// TIA Portal V20 export
VAR_GLOBAL   // PLC tag table "ENTRANCE"
   btnEmStopCraneEntCUCh1 AT %I500.0 : Bool;   // Emergency stop Crane entrance control panel Channel 1
   craneEntCUCraneOnKeyCh1 AT %I500.1 : Bool;   // Crane ON key switch Crane entrance control panel Channel 1
   mhOverloadBypassKeyCh1 AT %I500.2 : Bool;   // MH overload bypass key switch Channel 1
   craneMovementsProhibitionCh1 AT %I500.3 : Bool;   // Crane movements prohibition switch Channel 1
   btnEmStopCraneEntCUCh2 AT %I500.4 : Bool;   // Emergency stop Crane entrance control panel Channel 2
   craneEntCUCraneOnKeyCh2 AT %I500.5 : Bool;   // Crane ON key switch Crane entrance control panel Channel 2
   mhOverloadBypassKeyCh2 AT %I500.6 : Bool;   // MH overload bypass key switch Channel 2
   craneMovementsProhibitionCh2 AT %I500.7 : Bool;   // Crane movements prohibition switch Channel 2
   btnEmStopCraneEntCUCh1VS AT %I501.0 : Bool;   // Emergency stop Crane entrance control panel Channel 1 Supply
   craneEntCUCraneOnKeyCh1VS AT %I501.1 : Bool;   // Crane ON key switch Crane entrance control panel Channel 1 Supply
   mhOverloadBypassKeyCh1VS AT %I501.2 : Bool;   // MH overload bypass key switch Channel 1 Supply
   craneMovementsProhibitionCh1VS AT %I501.3 : Bool;   // Crane movements prohibition switch Channel 1 Supply
   btnEmStopCraneEntCUCh2VS AT %I501.4 : Bool;   // Emergency stop Crane entrance control panel Channel 2 Supply
   craneEntCUCraneOnKeyCh2VS AT %I501.5 : Bool;   // Crane ON key switch Crane entrance control panel Channel 2 Supply
   mhOverloadBypassKeyCh2VS AT %I501.6 : Bool;   // MH overload bypass key switch Channel 2 Supply
   craneMovementsProhibitionCh2VS AT %I501.7 : Bool;   // Crane movements prohibition switch Channel 2 Supply
   craneEntCUOpModeRCOS AT %I550.0 : Bool;   // Crane entrance control panel Operation mode RCOS
   craneEntCUOpModeCabin AT %I550.1 : Bool;   // Crane entrance control panel Operation mode Cabin
   craneEntCUOpModeRadio AT %I550.2 : Bool;   // Crane entrance control panel Operation mode Radio station
   craneEntCUOpModeGround AT %I550.3 : Bool;   // Crane entrance control panel Operation mode Ground level control
   craneEntCUOpModeSpare AT %I550.4 : Bool;   // Crane entrance control panel Operation mode Spare
   craneEntCUCraneOn AT %I550.5 : Bool;   // Crane entrance control panel Crane ON
   craneEntCUCraneOff AT %I550.6 : Bool;   // Crane entrance control panel Crane OFF
   craneEntCUFaultReset AT %I550.7 : Bool;   // Crane entrance control panel Fault reset
   craneEntCULampTest AT %I551.0 : Bool;   // Crane entrance control panel Lamp test
   craneEntCULtLeftLowSpeed AT %I551.1 : Bool;   // Crane entrance control panel LT left Low speed
   craneEntCULtLeftFullSpeed AT %I551.2 : Bool;   // Crane entrance control panel LT left Full speed
   craneEntCULtRightLowSpeed AT %I551.3 : Bool;   // Crane entrance control panel LT right Low speed
   craneEntCULtRightFullSpeed AT %I551.4 : Bool;   // Crane entrance control panel LT right Full speed
   craneEntCURailClampsOff AT %I551.5 : Bool;   // Crane entrance control panel Rail clamps OFF
   craneEntCURailClampsOn AT %I551.6 : Bool;   // Crane entrance control panel Rail clamps ON
   "spare(10)" AT %I551.7 : Bool;   // Spare
   cbCraneEntranceMainCtrlCabinetHeater AT %I552.0 : Bool;   // Crane entrance main control cabinet heater CB Feedback
   "spare(11)" AT %I552.1 : Bool;   // Spare
   "spare(12)" AT %I552.2 : Bool;   // Spare
   "spare(13)" AT %I552.3 : Bool;   // Spare
   "spare(14)" AT %I552.4 : Bool;   // Spare
   "spare(15)" AT %I552.5 : Bool;   // Spare
   "spare(16)" AT %I552.6 : Bool;   // Spare
   "spare(17)" AT %I552.7 : Bool;   // Spare
   indCraneEntCUMainsOK AT %Q550.0 : Bool;   // Crane entrance control panel 400V supply (indication)
   indCraneEntCUMLCStarted AT %Q550.1 : Bool;   // Crane entrance control panel Line contactor ON (indication)
   indCraneEntCUFault AT %Q550.2 : Bool;   // Crane entrance control panel Fault (indication)
   indCraneEntCULTReady AT %Q550.3 : Bool;   // Crane entrance control panel LT Ready (indication)
   indCraneEntCULTFault AT %Q550.4 : Bool;   // Crane entrance control panel LT Faut (indication)
   indCraneEntCURCOSActive AT %Q550.5 : Bool;   // Crane entrance control panel RCOS operation (indication)
   indCraneEntCURadioActive AT %Q550.6 : Bool;   // Crane entrance control panel Radio control operation (indication)
   indCraneEntCURailClampsOFF AT %Q551.0 : Bool;   // Crane entrance control panel Rail clamps OFF (indication)
   indCraneEntCURailClampsON AT %Q551.1 : Bool;   // Crane entrance control panel Rail clamps ON (indication)
   Tag_10 AT %Q551.2 : Bool;   // Spare
   Tag_11 AT %Q551.3 : Bool;   // Spare
   Tag_12 AT %Q551.4 : Bool;   // Spare
   Tag_13 AT %Q551.5 : Bool;   // Spare
   Tag_14 AT %Q551.6 : Bool;   // Spare
   Tag_15 AT %Q551.7 : Bool;   // Spare
END_VAR
